(*

short summary
=================
| This class provides assert statements for date and time types with 32 bit length
| It implements the interface :ref:`ISimpleDateAndTimeAssertions`
| For date and time (``DT``) use :ref:`SimpleDateAndTimeAssertions.dateAndTime`
| For date (``DATE``) use  :ref:`SimpleDateAndTimeAssertions.dateOnly`
| For time of day (``TOD``) use  :ref:`SimpleDateAndTimeAssertions.timeOfDay`

.. <legal notes>

legal notes
=================
| SPDX-FileCopyrightText: © 2022 ekvip automation GmbH <info@ekvip.de>
| SPDX-License-Identifier: Apache-2.0
| For details check: Apache-2.0_

.. _Apache-2.0: https://www.apache.org/licenses/LICENSE-2.0

.. </legal notes>

methods and properties
=======================

*)

{attribute 'reflection'}
FUNCTION_BLOCK INTERNAL SimpleDateAndTimeAssertions 
EXTENDS CNM_AbstractObject.Object
IMPLEMENTS ISimpleDateAndTimeAssertions, IAssertCallBacksetter
VAR
	(* class to handle date assertions *)
	dateAssertions		:DateAssertions32Bit();
	(* class to handle date and time assertions *)
	dateTimeAssertions	:DateTimeAssertions32Bit();
	(* class to handle time of day assertions *)
	timeOfDayAssertions	:TimeOfDayAssertions32Bit();
END_VAR

(*

short summary
=================
This abstract property returns the class name of the concrete object, 
It's for debugging purpose

.. <legal notes>

legal notes
=================
| SPDX-FileCopyrightText: © 2022 ekvip automation GmbH <info@ekvip.de>
| SPDX-License-Identifier: Apache-2.0
| For details check: Apache-2.0_

.. _Apache-2.0: https://www.apache.org/licenses/LICENSE-2.0

.. </legal notes>

*)

PROPERTY className :CNM_AbstractObject.ClassName
GET
className := 'CNM_AssertionInterfaceLib.SimplyDateAndTimeAssertions';
END_GET
END_PROPERTY

(*

short summary
=================
Returns the interface :ref:`I32BitDtAssertions`
with assert statements for 32 bit date and time ``DT``

.. <legal notes>

legal notes
=================
| SPDX-FileCopyrightText: © 2022 ekvip automation GmbH <info@ekvip.de>
| SPDX-License-Identifier: Apache-2.0
| For details check: Apache-2.0_

.. _Apache-2.0: https://www.apache.org/licenses/LICENSE-2.0

.. </legal notes>

*)

PROPERTY dateAndTime :I32BitDtAssertions
GET
dateAndTime := THIS^.dateTimeAssertions;
END_GET
END_PROPERTY

(*

short summary
=================
Returns the interface :ref:`I32BitDateAssertions`
with assert statements for 32 bit date ``DATE``

.. <legal notes>

legal notes
=================
| SPDX-FileCopyrightText: © 2022 ekvip automation GmbH <info@ekvip.de>
| SPDX-License-Identifier: Apache-2.0
| For details check: Apache-2.0_

.. _Apache-2.0: https://www.apache.org/licenses/LICENSE-2.0

.. </legal notes>

*)

PROPERTY dateOnly : I32BitDateAssertions
GET
dateOnly := THIS^.dateAssertions;
END_GET
END_PROPERTY

(*

short summary
=================
This methods is the setter for the callback class if an assertion was false

.. <legal notes>

legal notes
=================
| SPDX-FileCopyrightText: © 2022 ekvip automation GmbH <info@ekvip.de>
| SPDX-License-Identifier: Apache-2.0
| For details check: Apache-2.0_

.. _Apache-2.0: https://www.apache.org/licenses/LICENSE-2.0

.. </legal notes>

parameters
=================

*)

METHOD setCallBack
VAR_INPUT
	(* the class that must be informed if an assertion is false *)
	callBack	:IAssertCallback;  
END_VAR
THIS^.dateAssertions.setCallBack(callBack);
THIS^.dateTimeAssertions.setCallBack(callBack);
THIS^.timeOfDayAssertions.setCallBack(callBack);
END_METHOD

(*

short summary
=================
Returns the interface :ref:`I32BitDateAssertions`
with assert statements for 32 bit time of day ``TOD``

.. <legal notes>

legal notes
=================
| SPDX-FileCopyrightText: © 2022 ekvip automation GmbH <info@ekvip.de>
| SPDX-License-Identifier: Apache-2.0
| For details check: Apache-2.0_

.. _Apache-2.0: https://www.apache.org/licenses/LICENSE-2.0

.. </legal notes>

*)

PROPERTY timeOfDay :I32BitTodAssertions
GET
timeOfDay := THIS^.timeOfDayAssertions;
END_GET
END_PROPERTY

END_FUNCTION_BLOCK

(* stored: Version 1.1.0.1, ProductVersion 3.1.4024.11
   POU SimpleDateAndTimeAssertions: Id {f3dc97fb-181e-402c-8292-4576bcf882dc}, SpecialFunc None
   Property className: Id {b832bafb-84d2-4b1e-adf6-f14116155244}
   Get Get: Id {5015335e-ab46-4bf3-8221-71f22a741318}
   Property dateAndTime: Id {bb67ca2a-d53b-4d0e-9f82-b9aa54727ecf}
   Get Get: Id {437387f1-43e6-46c7-b9a6-f783d40a7537}
   Property dateOnly: Id {abb540b7-37c0-4d0f-bdf8-fb8b025068f2}
   Get Get: Id {b7a4fcbd-cc90-4002-ae5e-175383967ecd}
   Method setCallBack: Id {55c7dbf2-73b8-4a27-9087-f94699962405}
   Property timeOfDay: Id {1ba11a9a-0e79-4afb-aac9-e7d98b447f29}
   Get Get: Id {c913bd6b-1f4d-4c9a-8c5a-5788475d17a6} *)
